Fanuc KAREL source: kc00016.KL

-- PROVISIONAL review KL for V940-1; original PC SHA256 c9d256edd702d69b2e6721f048dbff7fd619930046d19d85b9023b4d77efee0b
-- Incomplete behavior may be omitted. Consult companion uncertainty JSON. Do not deploy.
PROGRAM KC00016
%NOLOCKGROUP
BEGIN
  -- V9_ZERO_TABLE_METADATA_HINT layout=0002_ascii; no indexed target words; source/name/runtime held
  -- UNRESOLVED_PC offsets 5-15; opcodes 27,22,31
  -- UNRESOLVED_PC offsets 20-24; opcodes 7F
END KC00016
